TYPE ST_CommunicatorData :
STRUCT
	stMessage					: ST_CommunicatorMassege;
	itfSender					: ITF_MessengerSender;
	arritfRecipient				: ARRAY [1..GVL_BaseConstans.MAX_NUMBER_OF_CLIENTS] OF ITF_MessengerRecipient;
	arrConfirmations			: ARRAY [1..GVL_BaseConstans.MAX_NUMBER_OF_CLIENTS] OF BOOL;		//potwierdzenia
	iNumberOfConfirmations		: INT;	//ilosc odbiorcow ktorzy musza potwierdzic
	iNumberOfRecipient			: INT;
END_STRUCT
END_TYPE

(* stored: Version 1.1.0.1
   DUT ST_CommunicatorData: Id {0658a430-f7e5-0cb0-25bf-a6b6e5b94e0d} *)
